{attribute addProperty BoxType "KL2212"}
{attribute addProperty Id "Channel_1Channel_9147928600Channel_2Channel_9147928600"}
{attribute addProperty CRC "2776897432"}
{attribute addProperty SizeInBites "0"}
{attribute addProperty SizeInBytes "0"}
TYPE KL2212_A5841798 :
STRUCT
	{attribute addProperty Name "Channel_1"}
	Channel_1 : Channel_91479286;
	{attribute addProperty Name "Channel_2"}
	Channel_2 : Channel_91479286;
END_STRUCT
END_TYPE

(* stored: Version 1.2.0.0, ProductVersion 3.1.4024.9
   DUT KL2212_A5841798: Id {93678b01-873f-4407-ae10-bf52aa18df22} *)
